// TIA Portal V19 export
DATA_BLOCK "PPrgArchive2"   // DB519
// stored: IsOnlyStoredInLoadMemory true, MemoryReserve 0, Namespace G
   VAR RETAIN
      PRG : Array[101..200] of "PPrg_Data";
   END_VAR
BEGIN
END_DATA_BLOCK
